FUNCTION_BLOCK SS4_v_direct_V2 (* Composite FB wrapping other FBs *)
  (* Standard: 61499-2 *)
  (* Version 1.0, 2024-10-03, DEVIASH *)
  PACKAGE UserLibs::SubStations::SS4;
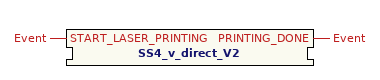
  EVENT_INPUT
    START_LASER_PRINTING; (* Initialization Request *)
  END_EVENT
  EVENT_OUTPUT
    PRINTING_DONE; (* Initialization Confirm *)
  END_EVENT
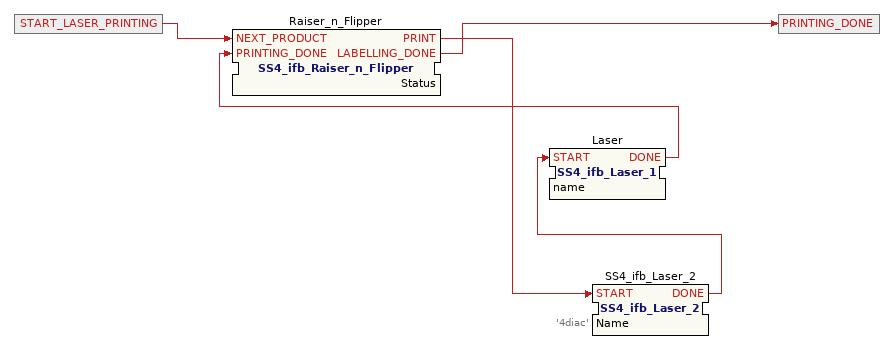
  FBS
    Raiser_n_Flipper : SS4_ifb_Raiser_n_Flipper;
    Laser : SS4_ifb_Laser_1;
    SS4_ifb_Laser_2 : SS4_ifb_Laser_2(Name := '4diac');
  END_FBS
  EVENT_CONNECTIONS
    START_LASER_PRINTING TO Raiser_n_Flipper.NEXT_PRODUCT;
    Raiser_n_Flipper.LABELLING_DONE TO PRINTING_DONE;
    Raiser_n_Flipper.PRINT TO SS4_ifb_Laser_2.START;
    SS4_ifb_Laser_2.DONE TO Laser.START;
    Laser.DONE TO Raiser_n_Flipper.PRINTING_DONE;
  END_CONNECTIONS
END_FUNCTION_BLOCK
